/// This function block is a container for all I/Os that are used by this unit.
/// The parent of all objects can be directly transfered in their constructor (this is only relevant for equipment objects
/// that have to be managed (e.g. [DebouncedInput](xref:ZEquipment.DebouncedInput), [Light](xref:ZEquipment.Light), ...).
FUNCTION_BLOCK DrillingIo EXTENDS DrillingContainer
VAR
  {attribute 'hide'}
  _iobridge : ZApplication.IoBridge(_parent);
END_VAR
VAR_INPUT

{attribute '__ZwPlcUnitEquipmentDeclaration__'} // Do not remove this attribute! It is used for code generation.
END_VAR

IF _isInitialized
THEN
  RETURN;
END_IF

  _iobridge.SetLogger(_parent._logger);

{attribute '__ZwPlcUnitEquipmentImplementation__'} // Do not remove this attribute! It is used for code generation.

_isInitialized := TRUE;

END_FUNCTION_BLOCK

(* stored: Version 1.1.0.1
   POU DrillingIo: Id {135c2d33-9695-485f-b707-123355615597}, SpecialFunc None *)
